// TIA Portal V17 export
// export: Created 2026-04-13T11:12:03.5986543Z, ExportSetting WithDefaults, DisplayName Totally Integrated Automation Portal, DisplayVersion V17 Update 4, DisplayName TIA Portal Openness, DisplayVersion V17 Update 4, DisplayName TIA Portal Version Control Interface, DisplayVersion V17, DisplayName SINAMICS Startdrive Advanced, DisplayVersion V17, DisplayName SINAMICS Startdrive G130, G150, S120, S150, SINAMICS MV, S210, DisplayVersion V17, DisplayName SINAMICS Startdrive G110M, G120, G120C, G120D, G120P, G115D, DisplayVersion V17, DisplayName STEP 7 Professional, DisplayVersion V17 Update 4, DisplayName STEP 7 Safety, DisplayVersion V17, DisplayName WinCC Professional, DisplayVersion V17 Update 4
FUNCTION "0- IO Configure" : Void   // FC10, LAD
TITLE = 1_IO Configure
{ S7_Optimized_Access := 'TRUE' }
VERSION : 0.1
// stored: AutoNumber true, IsIECCheckEnabled false, SetENOAutomatically false, UDAEnableTagReadback false
BEGIN

REGION Network 1 (SCL): IJT急停
   //DI/DO地址分配-----------------------------------------------------------------------
   //"SV".JF进风加热比例调节阀
   //"MYH氧含仪隔断阀"
   //"AWQ尾气温度高高报"
   //"AYJ一级排液阀开报警"



   "ISF送风机" := NOT "I0.0";
   "IYF引风机" := NOT "I0.1";
   "ILX离心雾化器" := NOT "I0.2";
   "IJL进料泵" := "I0.3";
   "IDJ电加热" :=  "I0.4";
   "ISF输送风机" := "I0.5";
   "ISF输送加热" := "I0.6";
   "IJT急停" := "I0.7";

   "ILQ冷却水流量" := "I1.0";
   "ILD冷冻水流量" := "I1.1";
   "IJF进风冷却水流量" := "I1.2";
   "IPY排液流量" := "I1.3";
   "IBD补氮阀开反馈" := "I1.4";
   "IBD补氮阀关反馈" := "I1.5";
   "IJD进氮阀开反馈" := "I1.6";
   "IJD进氮阀关反馈" := "I1.7";

   "IXY泄压阀开反馈" := "I2.0";
   "IXY泄压阀关反馈" := "I2.1";
   "IQL气流雾化阀开反馈" := "I2.2";
   "IQL气流雾化阀关反馈" := "I2.3";
   "ISF输送进风阀开反馈" := "I2.4";
   "ISF输送进风阀关反馈" := "I2.5";
   "IKS开式排风隔断阀开反馈" := "I2.6";
   "IKS开式排风隔断阀关反馈" := "I2.7";

   "IBS闭式排风隔断阀开反馈" := "I3.0";
   "IBS闭式排风隔断阀关反馈" := "I3.1";
   "IKS开式进风隔断阀开反馈" := "I3.2";
   "IKS开式进风隔断阀关反馈" := "I3.3";
   "IBS闭式进风隔断阀开反馈" := "I3.4";
   "IBS闭式进风隔断阀关反馈" := "I3.5";
   "IYJ一级冷却水阀开反馈" := "I3.6";
   "IYJ一级冷却水阀关反馈" := "I3.7";

   "IEJ二级冷冻水阀开反馈" := "I4.0";
   "IEJ二级冷冻水阀关反馈" := "I4.1";
   "IYJ一级排液阀开反馈" := "I4.2";
   "IYJ一级排液阀关反馈" := "I4.3";
   "IEJ二级排液阀开反馈" := "I4.4";
   "IEJ二级排液阀关反馈" := "I4.5";
   "ICW除雾排液阀开反馈" := "I4.6";
   "ICW除雾排液阀关反馈" := "I4.7";

   "IRJ溶剂回收排放阀开反馈" := "I5.0";
   "IRJ溶剂回收排放阀关反馈" := "I5.1";
   "IJF进风冷却水阀开反馈" := "I5.3";
   "IJF进风冷却水阀关反馈" := "I5.2";

   "ITD塔顶清洗球阀开反馈" := "I5.4";
   "ITD塔顶清洗球阀关反馈" := "I5.5";

   "IQX清洗伸缩气缸升反馈" := "I5.6";//升
   "IQX清洗伸缩气缸降反馈" := "I5.7";//降

   "IJF进风保护温度" := "I6.0";
   "ISS输送保护温度" := "I6.1";
   "IBP爆破片1反馈" := NOT "I6.2";
   "IBP爆破片2反馈" := NOT "I6.3";
   "ISN室内排水开反馈" := "I6.7";
   "ISN室内排水关反馈" := "I6.6";
   "IRJ溶剂排液泵开反馈" := "I6.4";
   "IRJ溶剂排液泵关反馈" := "I6.5";

   (* 冷却水流量开关报警
   冷冻水流量开关报警
   进风冷却水流量开关报警
   排液流量开关报警
    电加热故障
   输送风机故障
   输送加热故障
   爆破片1故障
   爆破片2故障

   *)
   "AQX清洗伸缩气缸关报警" := 0;
   "AQX清洗伸缩气缸开报警" := 0;

   (* IF "ILQ冷却水流量" THEN
       "ALQ冷却水流量低报警" := 1;
   ELSE
       "ALQ冷却水流量低报警" := 0;
   END_IF;

   IF "ILD冷冻水流量" THEN
       "ALD冷冻水流量低报警" := 1;
   ELSE
       "ALD冷冻水流量低报警" := 0;
   END_IF; *)

   IF "IJF进风冷却水流量" THEN
       "AJF进风冷却水流量低报警" := 1;
   ELSE
       "AJF进风冷却水流量低报警" := 0;
   END_IF;

   //暂时注销掉
   (* IF "IPY排液流量" THEN
       "APY排液流量低报警" := 1;
   ELSE
       "APY排液流量低报警" := 0;
   END_IF; *)

   IF "IBP爆破片1反馈" THEN
       "ABP爆破片1反馈报警" := 1;
   ELSE
       "ABP爆破片1反馈报警" := 0;
   END_IF;

   IF "IBP爆破片2反馈" THEN
       "ABP爆破片2反馈报警" := 1;
   ELSE
       "ABP爆破片2反馈报警" := 0;
   END_IF;

   IF "IDJ电加热" THEN
       "ADJ电加热报警" := 1;
   ELSE
       "ADJ电加热报警" := 0;
   END_IF;

   IF "ISF输送风机" THEN
       "ASF输送风机故障报警" := 1;
   ELSE
       "ASF输送风机故障报警" := 0;
   END_IF;


   IF "ISF输送加热" THEN
       "ASF输送加热故障报警" := 1;
   ELSE
       "ASF输送加热故障报警" := 0;
   END_IF;

   IF NOT "IJT急停" THEN
       "AJT急停报警" := 1;
   ELSE
       "AJT急停报警" := 0;
   END_IF;
   (* IF ILQ冷却水流量开关
   冷冻水流量开关报警
   进风冷却水流量开关报警
   排液流量开关报警
   电加热故障
   输送风机故障
   输送加热故障
   爆破片1故障
   爆破片2故障 *)

   "Q0.0" := "QSF送风机";
   "Q0.1" := "QSF送风机风扇";
   "Q0.2" := "QYF引风机";
   "Q0.3" := "QYF引风机风扇";
   "Q0.4" := "QLX离心雾化";
   "Q0.5" := "QLX离心雾化风扇";
   "Q0.6" := "QLX离心雾化油泵";
   "Q0.7" := "QJL进料泵";

   "Q1.0" := "QJL进料泵风扇";
   "Q1.1" := "QDJ电加热器";
   "Q1.2" := "QSS输送风机";
   "Q1.3" := "QSS输送加热器";
   "Q1.4" := "QFM蜂鸣器";
   "Q1.5" := "QZS指示灯";
   "Q1.6" := "QYS钥匙开关";
   "Q1.7" := "QZM照明灯";

   "Q2.0" := "QBY备用1";
   "Q2.1" := "QCC除尘脉冲";
   "Q2.2" := "QBY备用2";
   "Q2.3" := "QBY备用3";
   "Q2.4" := "QBY备用4";
   "Q2.5" := "QRS热水洗请求";
   "Q2.6" := 0;//无
   "Q2.7" := "QBY备用7";

   "Q3.0" := "QXY泄压阀";
   "Q3.1" := "QJF进风冷却水阀";
   "Q3.2" := "QSS输送进风阀";
   "Q3.3" := "QQL气流雾化阀";
   "Q3.4" := "QKS开式排风隔断阀";
   "Q3.5" := "QBS闭式排风隔断阀";
   "Q3.6" := "QKS开式进风隔断阀";
   "Q3.7" := "QBS闭式进风隔断阀";

   "Q4.0" := "QYJ一级冷却水阀";
   "Q4.1" := "QEJ二级冷冻水阀";
   "Q4.2" := "QYJ一级排液阀";
   "Q4.3" := "QEJ二级排液阀";
   "Q4.4" := "QCW除雾排液阀";
   "Q4.5" := "QRJ溶剂回收排放阀";
   "Q4.6" := "QSN室内排水隔膜泵";//回程泵
   "Q4.7" := "QRJ溶剂排液泵";

   "Q5.0" := "QBY备用10";;
   "Q5.1" := "QBY备用11";;
   "Q5.2" := "QASA室内回水阀";//振打
   "Q5.3" := "QBD补氮阀";
   "Q5.4" := "QASA室外回水阀";//振打
   "Q5.5" := "QJD进氮阀";
   "Q5.6" := "QCC除尘气锤1";
   "Q5.7" := "QCC除尘气锤2";

   "Q6.0" := "QTD塔顶清洗球阀";//加阀岛
   "Q6.1" := "QRJ溶剂排液泵进阀";
   "Q6.3" := "QSB设备振打";
   //阀导
   "Q10.0" := "QSN室内清洗总阀"; //室内清洗总阀
   "Q10.1" := "QASA室内回水阀";//A室内回水阀
   "Q10.2" := "QASA室外回水阀";//A室外回水阀
   "Q10.3" := "QJF进风蒸汽开关阀";
   "Q10.4" := "QJF进风蒸汽排水阀";
   "Q10.5" := "QLG料罐清洗阀";
   "Q10.6" := "QQX清洗溶剂出阀";
   "Q10.7" := "QWL物料进阀";

   "Q11.0" := "QYJ一级出料上阀";
   "Q11.1" := "QYJ一级出料下阀";
   "Q11.2" := "QEJ二级出料上阀";
   "Q11.3" := "QEJ二级出料下阀";
   "Q11.4" := "QCC除尘出料上阀";
   "Q11.5" := "QCC除尘出料下阀";
   "Q11.6" := "QHF回风蒸汽开关阀";
   "Q11.7" := "QHF回风蒸汽排水阀";

   "Q12.0" := "QSS输送出料上阀";
   "Q12.1" := "QSS输送出料下阀";//空的，未接
   "Q12.2" := "QQG气缸升";
   "Q12.3" := "QQG气缸降";
   "Q12.4" := "QZT主塔清洗进水阀";
   "Q12.5" := "QXF旋风管道清洗阀";
   "Q12.6" := "QYJ一级旋风清洗阀";
   "Q12.7" := "QEJ二级旋风清洗阀";

   "Q13.0" := "QCC除尘管道清洗阀";
   "Q13.1" := "QCC除尘清洗阀";
   "Q13.2" := "QSS输送管路清洗阀";
   "Q13.3" := "QLC料仓清洗阀";
   "Q13.4" := "QJR加热清洗阀";
   "Q13.5" := "QWK蜗壳清洗阀";//Q6.0
   "Q13.6" := "QCF出风高效清洗阀";
   "Q13.7" := "QZT主塔排水阀";

   "Q14.0" := "QSS输送管路排水阀";
   "Q14.1" := "QLC料仓清洗排水阀";
   "Q14.2" := "QSF送风机清洗阀";
   "Q14.3" := "QYF引风机清洗阀";
   "Q14.4" := "QYJ一级冷凝清洗阀";
   "Q14.5" := "QEJ二级冷凝清洗阀";
   "Q14.6" := "QSF送风机排水阀";
   "Q14.7" := "QYF引风机排水阀";

   "Q15.0" :="QYJ一级旋风振打锤" ;//主塔振打1
   "Q15.1" :="QYJ一级旋风振荡器" ;//主塔振打2
   "Q15.2" := "QEJ二级旋风振打锤";//主塔振打3
   "Q15.3" :="QZT主塔气锤4" ;//主塔振打4
   "Q15.4" :="QQZ前置水阀" ;//布袋振打1
   //"Q15.5" :="QSB设备振打" ;//布袋振打2
   (* "Q15.6" :="QBD布袋振打3" ;//布袋振打3
   "Q15.7" :="QBD布袋振打4" ;//布袋振打4 *)

   "Q15.6" :="QYH氧含仪隔断阀" ;//氧含仪隔断阀1
   "Q15.7" :="QHS回水隔断阀1" ;//这个空的



   //QW

   "QW100" := "QWFK放空比例调节阀";
   "QW102" := "QWJF进风加热比例调节阀";
   "QW104" := "QWHF回风加热比例调节阀";

   "QW108" := "QWSF送风机";
   "QW110" := "QWYF引风机";
   "QW112" := "QWLX离心雾化器";
   "QW114" := "QWJL进料泵";


   //IW 

   "IWJF进风流量计" := "IW100";
   "IWJL进料流量" := "IW102";
   "IWJF进风压差变送器" := "IW104";
   "IWCF出风高效压差变送器" := "IW106";

   "IWBD布袋压差变送器" := "IW108";
   "IWSS输送高效压差变送器" := "IW110";
   "IWJL进料压力" := "IW112";
   "IWTN塔内压力" := "IW114";

   "IWGD管道压力变送器" := "IW116";
   "IWJD进氮压力" := "IW118";
   "IWFK放空比例反馈" := "IW120";
   "IWJF进风加热比例反馈" := "IW122";

   "IWHF回风加热比例反馈" := "IW124";
   "IWWH雾化油压" := "IW126";
   "IWYH氧含仪1" := "IW128";
   "IWYH氧含仪2" := "IW130";

   //第二个模块
   "IWYJ一级溶剂液位计" := "IW132";
   "IWEJ二级溶剂液位计" := "IW134";
   "IWCW除雾溶剂液位计" := "IW136";
   "IWFD阀岛气压" := "IW138";

   "IWQZ前置水罐液位计" := "IW140";
   "IWBY备用2" := "IW142";
   "IWBY备用3" := "IW144";
   "IWBY备用4" := "IW146";


   //IW140-IW146空。
   "IWBY备用5" := "IW148";
   "IWSF送风机" := "IW150";
   "IWYF引风机" := "IW152";
   "IWLX离心雾化器" := "IW154";

   "IWJL进料泵" := "IW156";
   "IWBY备用6" := "IW158";
   "IWBY备用7" := "IW160";
   "IWBY备用8" := "IW162";
END_REGION
END_FUNCTION
